PROGRAM MAIN
VAR
END_VAR

P_SMI();

END_PROGRAM

(* stored: Version 1.1.0.1, ProductVersion 3.1.4024.0
   POU MAIN: Id {bf0efed6-bfb2-4408-97ec-71af699189ec}, SpecialFunc None *)
